PROGRAM MAIN
VAR
	READ  : INT;
	WRITE : INT;
END_VAR

READ := read +1 ;

END_PROGRAM

(* stored: Version 1.1.0.1, ProductVersion 3.1.4024.12
   POU MAIN: Id {163b8446-4c09-4e0f-b4e3-176ceac5542f}, SpecialFunc None *)
